SUBAPPLICATION Uebung_051 (* DigitalInput_I1-_I4 auf DigitalOutput_Q1-_Q4 *)
  (* Standard: 61499-2 *)
  (* Version 1.0, 2023-10-23, franz *)
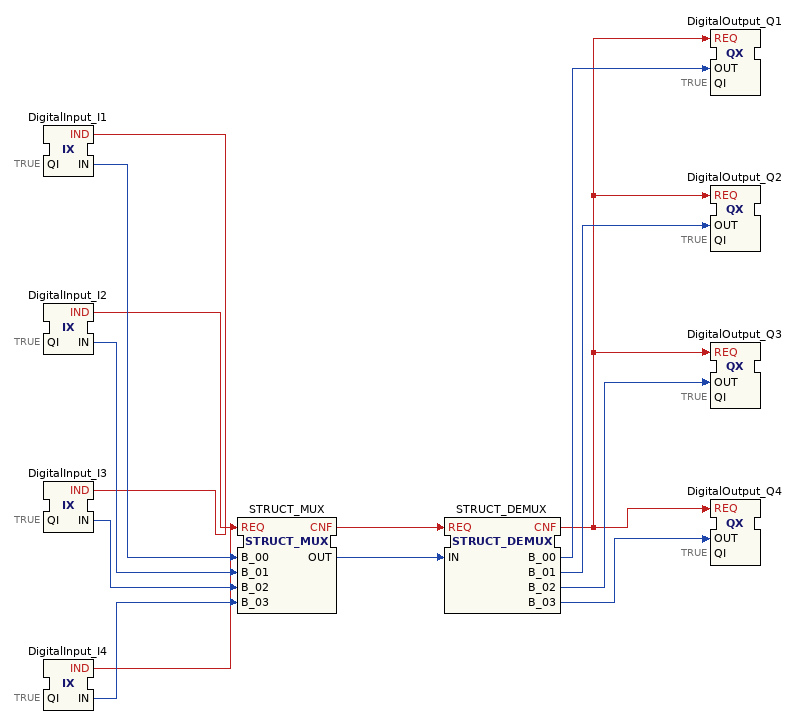
  FBS
    DigitalOutput_Q1 : QX(QI := TRUE);
    DigitalInput_I1 : IX(QI := TRUE);
    DigitalOutput_Q2 : QX(QI := TRUE);
    DigitalInput_I2 : IX(QI := TRUE);
    DigitalOutput_Q3 : QX(QI := TRUE);
    DigitalInput_I3 : IX(QI := TRUE);
    DigitalOutput_Q4 : QX(QI := TRUE);
    DigitalInput_I4 : IX(QI := TRUE);
    STRUCT_DEMUX : STRUCT_DEMUX; {SET_ATTRIBUTE(StructuredType, ST04B)}
    STRUCT_MUX : STRUCT_MUX; {SET_ATTRIBUTE(StructuredType, ST04B)}
  END_FBS
  EVENT_CONNECTIONS
    DigitalInput_I1.IND TO STRUCT_MUX.REQ;
    DigitalInput_I2.IND TO STRUCT_MUX.REQ;
    DigitalInput_I3.IND TO STRUCT_MUX.REQ;
    DigitalInput_I4.IND TO STRUCT_MUX.REQ;
    STRUCT_MUX.CNF TO STRUCT_DEMUX.REQ;
    STRUCT_DEMUX.CNF TO DigitalOutput_Q1.REQ;
    STRUCT_DEMUX.CNF TO DigitalOutput_Q2.REQ;
    STRUCT_DEMUX.CNF TO DigitalOutput_Q3.REQ;
    STRUCT_DEMUX.CNF TO DigitalOutput_Q4.REQ;
  END_CONNECTIONS
  DATA_CONNECTIONS
    DigitalInput_I1.IN TO STRUCT_MUX.B_00;
    DigitalInput_I2.IN TO STRUCT_MUX.B_01;
    DigitalInput_I3.IN TO STRUCT_MUX.B_02;
    DigitalInput_I4.IN TO STRUCT_MUX.B_03;
    STRUCT_MUX.OUT TO STRUCT_DEMUX.IN;
    STRUCT_DEMUX.B_00 TO DigitalOutput_Q1.OUT;
    STRUCT_DEMUX.B_01 TO DigitalOutput_Q2.OUT;
    STRUCT_DEMUX.B_02 TO DigitalOutput_Q3.OUT;
    STRUCT_DEMUX.B_03 TO DigitalOutput_Q4.OUT;
  END_CONNECTIONS
END_SUBAPPLICATION
